// TIA Portal V19 export
DATA_BLOCK "Drucktest"   // DB340
{ S7_Optimized_Access := 'FALSE' }
// stored: AutoNumber false
   VAR RETAIN
      akt_Index : Int := 0;
      Index_Panel : Int;
      Ergebnis : Array[0..100] of Struct
         "Name" : String[12];
         Zeit : DTL;
         ok : Bool;
         Fehler : Bool;
      END_STRUCT;
   END_VAR
BEGIN
END_DATA_BLOCK
